PROGRAM MAIN
VAR
END_VAR

END_PROGRAM

(* stored: Version 1.1.0.1
   POU MAIN: Id {b33004eb-8057-44d3-a1ea-77f02b6b92b4} *)
